(* IEC 61131-3 sources: Industry-PLC-LLM/data/PLCBEAD_repo/PLCBEAD_PLCEmbed-main/PLC-BEAD/Source/GEB/AIN1, 1 file *)

(* ---- AIN1.ST ---- *)
FUNCTION_BLOCK AIN1

	VAR_INPUT
		IN :	DWORD;
		SIGN_BIT :	INT := 255;
		ERROR_BIT :	INT := 255;
		ERROR_CODE_EN :	BOOL := FALSE;
		ERROR_CODE :	DWORD;
		OVERFLOW_BIT :	INT := 255;
		OVERFLOW_CODE_EN :	BOOL;
		OVERFLOW_CODE :	DWORD;
		BIT_0 :	INT;
		BIT_N :	INT := 31;
		OUT_MIN :	REAL;
		OUT_MAX :	REAL := 10.0;
		CODE_MIN :	DWORD;
		CODE_MAX :	DWORD := DWORD#16#FFFFFFFF;
		ERROR_OUTPUT :	REAL;
		OVERFLOW_OUTPUT :	REAL := 10.0;
	END_VAR

	VAR_OUTPUT
		OUT :	REAL;
		SIGN :	BOOL;
		ERROR :	BOOL;
		OVERFLOW :	BOOL;
	END_VAR

	VAR
		tb :	DWORD;
	END_VAR

	ERROR := ((SHR(IN,ERROR_BIT) AND DWORD#16#0000_0001) = DWORD#1) OR (ERROR_CODE_EN AND ERROR_CODE = IN);
	IF ERROR THEN
		OUT := ERROR_OUTPUT;
		RETURN;
	END_IF;

	tb := SHR(SHL(IN, 31 - BIT_N), 31 - BIT_N + BIT_0);

	OVERFLOW := ((SHR(IN,OVERFLOW_BIT) AND DWORD#16#0000_0001) = DWORD#1) OR (OVERFLOW_CODE_EN AND OVERFLOW_CODE = IN) OR (tb < CODE_MIN OR tb > CODE_MAX);
	IF OVERFLOW THEN
		OUT := OVERFLOW_OUTPUT;
		RETURN;
	END_IF;

	SIGN := (SHR(IN,SIGN_BIT) AND DWORD#16#0000_0001) = DWORD#1;

	OUT := (UDINT_TO_REAL(DWORD_TO_UDINT(tb) - DWORD_TO_UDINT(CODE_MIN)) * (OUT_MAX - OUT_MIN) / UDINT_TO_REAL(DWORD_TO_UDINT(CODE_MAX) - DWORD_TO_UDINT(CODE_MIN)) + OUT_MIN);
	IF SIGN THEN OUT := OUT * -1.0; END_IF;

	(* extract ERROR bit *)
	ERROR := ((SHR(IN,ERROR_BIT) AND DWORD#16#0000_0001) = DWORD#1) OR (ERROR_CODE_EN AND ERROR_CODE = IN);
	IF ERROR THEN
		OUT := ERROR_OUTPUT;
		RETURN;
	END_IF;

	(* strip off the data input *)
	tb := SHR(SHL(IN, 31 - BIT_N), 31 - BIT_N + BIT_0);

	(* extract OVERFLOW bit *)
	OVERFLOW := ((SHR(IN,OVERFLOW_BIT) AND DWORD#16#0000_0001) = DWORD#1) OR (OVERFLOW_CODE_EN AND OVERFLOW_CODE = IN) OR (tb < CODE_MIN OR tb > CODE_MAX);
	IF OVERFLOW THEN
		OUT := OVERFLOW_OUTPUT;
		RETURN;
	END_IF;

	(* extract SIGN bit *)
	SIGN := (SHR(IN,SIGN_BIT) AND DWORD#16#0000_0001) = DWORD#1;

	(* convert IN to OUT *)
	OUT := (UDINT_TO_REAL(DWORD_TO_UDINT(tb) - DWORD_TO_UDINT(CODE_MIN)) * (OUT_MAX - OUT_MIN) / UDINT_TO_REAL(DWORD_TO_UDINT(CODE_MAX) - DWORD_TO_UDINT(CODE_MIN)) + OUT_MIN);
	IF SIGN THEN OUT := OUT * - 1.0; END_IF;

END_FUNCTION_BLOCK

PROGRAM program0
  VAR
	IN               :	DWORD;
	SIGN_BIT         :	INT ;
	ERROR_BIT        :	INT ;
	ERROR_CODE_EN    :	BOOL ;
	ERROR_CODE       :	DWORD;
	OVERFLOW_BIT     :	INT ;
	OVERFLOW_CODE_EN :	BOOL;
	OVERFLOW_CODE    :	DWORD;
	BIT_0            :	INT;
	BIT_N            :	INT;
	OUT_MIN          :	REAL;
	OUT_MAX          :	REAL ;
	CODE_MIN         :	DWORD;
	CODE_MAX         :	DWORD ;
	ERROR_OUTPUT     :	REAL;
	OVERFLOW_OUTPUT  :	REAL ;

	OUT      :	REAL;
	SIGN     :	BOOL;
	ERROR    :	BOOL;
	OVERFLOW :	BOOL;

	func_block : AIN1;
  END_VAR
	func_block.IN               :=IN              ;
	func_block.SIGN_BIT         :=SIGN_BIT        ;
	func_block.ERROR_BIT        :=ERROR_BIT       ;
	func_block.ERROR_CODE_EN    :=ERROR_CODE_EN   ;
	func_block.ERROR_CODE       :=ERROR_CODE      ;
	func_block.OVERFLOW_BIT     :=OVERFLOW_BIT    ;
	func_block.OVERFLOW_CODE_EN :=OVERFLOW_CODE_EN;
	func_block.OVERFLOW_CODE    :=OVERFLOW_CODE   ;
	func_block.BIT_0            :=BIT_0           ;
	func_block.BIT_N            :=BIT_N           ;
	func_block.OUT_MIN          :=OUT_MIN         ;
	func_block.OUT_MAX          :=OUT_MAX         ;
	func_block.CODE_MIN         :=CODE_MIN        ;
	func_block.CODE_MAX         :=CODE_MAX        ;
	func_block.ERROR_OUTPUT     :=ERROR_OUTPUT    ;
	func_block.OVERFLOW_OUTPUT  :=OVERFLOW_OUTPUT ;

	func_block();
	OUT     := func_block.OUT     ;
	SIGN    := func_block.SIGN    ;
	ERROR   := func_block.ERROR   ;
	OVERFLOW:= func_block.OVERFLOW;
END_PROGRAM
